// TwinCAT 3 PLC project Untitled1
// ProgramVersion: 3.1.4024.0
// libraries:
//   Tc2_Standard, * (Beckhoff Automation GmbH)
//   Tc2_System, * (Beckhoff Automation GmbH)
//   Tc2_Utilities, * (Beckhoff Automation GmbH)
//   Tc3_Module, * (Beckhoff Automation GmbH)
//   VisuDialogs, * (System)
// project tree:
//   DUTs/ E_PIZZA_TYPES.TcDUT, ST_PIZZA.TcDUT
//   / GlobalTextList.TcGTLO, PlcTask.TcTTO, Visualization Manager.TcVMO (not stored)
//   GVLs/ HMI_VARS.TcGVL
//   POUs/ FB_PizzaOven.TcPOU, F_FIFO_WRITE.TcPOU, MAIN.TcPOU
//   VISUs/ Visualization.TcVIS
// real-time tasks:
//   TASK PlcTask: cycle T#10ms, priority 20, ADS port 350

CONFIGURATION Untitled1
    RESOURCE PLC ON TwinCAT3
        TASK PlcTask(INTERVAL := T#10ms, PRIORITY := 20);
        PROGRAM MAIN WITH PlcTask : MAIN;
    END_RESOURCE
END_CONFIGURATION

// ---- DUTs/E_PIZZA_TYPES.TcDUT
{attribute 'qualified_only'}
{attribute 'strict'}
TYPE E_PIZZA_TYPES :
(
	eType_Cheese := 0,
	eType_Pepperoni := 1,
	eType_Olives := 2
);
END_TYPE

// ---- DUTs/ST_PIZZA.TcDUT
TYPE ST_PIZZA :
STRUCT
	bExist : BOOL;
	dtTimeEnteredOven : DT;
	dtTimeExitedOven : DT;
	tTimeInOven : TIME;
	eType : E_PIZZA_TYPES;	// 0 - cheese, 1 - pepperoni, 2 - olives
END_STRUCT
END_TYPE

// ---- GVLs/HMI_VARS.TcGVL
{attribute 'qualified_only'}
VAR_GLOBAL
	iState : DINT;
	bStartButton : BOOL;
	
	arrPizzaHistory : ARRAY[0..100] OF ST_PIZZA;	
	
	fbNT_GetTime: NT_GetTime;
	stCurrentTime : TIMESTRUCT;
	
END_VAR

// ---- POUs/MAIN.TcPOU
PROGRAM MAIN
VAR
	
	fbMyPizzaOven : ARRAY[0..MAX_OVENS] OF FB_PizzaOven;	// My instance of oven 1
	
	bLoadPizza : BOOL;	// Put a pizza on the input side
	bRemovePizza : BOOL;	// Take pizza off output side
	
	i : DINT;
	
	fbMyTimer : TON;
	
	fbNT_GetTime: NT_GetTime;

END_VAR

VAR CONSTANT
	MAX_OVENS : DINT := 1; // This is 2 because the array starts at 0
END_VAR

FOR i:= 0 TO MAX_OVENS DO
	fbMyPizzaOven[i](bLoadPizza:=bLoadPizza, bRemovePizza:=bRemovePizza);
END_FOR

fbMyTimer(IN:=NOT fbMyTimer.Q, PT:=T#100MS);

fbNT_GetTime(
	NETID := '',
	START := fbMyTimer.Q,
	TIMESTR => hmi_vars.stCurrentTime);

END_PROGRAM

// ---- POUs/FB_PizzaOven.TcPOU
FUNCTION_BLOCK FB_PizzaOven
VAR_INPUT
	
	bLoadPizza : BOOL;	// Put a pizza on the input side
	bRemovePizza : BOOL;	// Take pizza off output side

END_VAR
VAR_OUTPUT

	bBuzzer : BOOL;
	bLight : BOOL;

	iTotalPizzasCooked : UDINT;

END_VAR
VAR
	
	stCurrentTime : TIMESTRUCT;
	dtCurrentTime : DT;

	fbLoad_RTRIG : R_TRIG;
	fbRemove_RTRIG : R_TRIG;	

	stPizzaOnDeck : ST_PIZZA;	// Location of possible pizza
	stPizzaInOven : ST_PIZZA;
	stPizzaDone : ST_PIZZA;
	
	// timers
	fbMyTimer : TON;	// My timer... for stuff.

	iState : DINT;
	ILastState : DINT;
	sStateDesc : STRING;
	arrStateDescHistory : ARRAY[1..100] OF STRING;
	
	bStartButton: BOOL;
	arrPizzaHistory: BYTE;
	TIMESTR: STRING(INT#4);
END_VAR
VAR CONSTANT
	stNULL_PIZZA : ST_PIZZA;
END_VAR

dtCurrentTime := SYSTEMTIME_TO_DT(stCurrentTime);

// If there is room
IF stPizzaOnDeck.bExist AND NOT stPizzaInOven.bExist THEN
	stPizzaInOven := stPizzaOnDeck;
	stPizzaOnDeck := stNULL_PIZZA;	// Remove pizza
END_IF

fbLoad_RTRIG(clk := bLoadPizza);
IF fbLoad_RTRIG.Q THEN
	stPizzaOnDeck.bExist := TRUE;
	stPizzaOnDeck.eType := 2;	// Olives
END_IF

fbRemove_RTRIG(clk := bRemovePizza);
IF fbRemove_RTRIG.Q THEN
	//F_FIFO_WRITE(cbData := SIZEOF(stPizzaDone), pData := ADR(stPizzaDone),
	//				cbBuffer := SIZEOF(arrPizzaHistory), pBuffer := ADR(arrPizzaHistory)
	//);	//It gives an error for arrPizzaHistory, I don't know how to fix it
	stPizzaDone := stNULL_PIZZA;
END_IF

CASE iState OF
	0:	// Wait for pizza in oven
		sStateDesc := 'Waiting on pizza now.';
		IF stPizzaInOven.bExist THEN
			stPizzaInOven.dtTimeEnteredOven := dtCurrentTime;
			iState := 10;
		END_IF
	10:	// We just got a pizza!
		sStateDesc := 'Baking that pizza now.';
		fbMyTimer(IN:=TRUE, PT:=T#3S);
		
		IF fbMyTimer.Q THEN
			fbMyTimer(IN:=FALSE);
			iState := 20;
		END_IF
	20:	// Can we move the pizza out of the oven? It's going to burn!
		IF NOT stPizzaDone.bExist THEN
			// Simulate conveyor
			stPizzaInOven.dtTimeExitedOven := dtCurrentTime;
			stPizzaDone := stPizzaInOven;
			stPizzaInOven := stNULL_PIZZA;
			bBuzzer := FALSE;
			iState := 30;
		ELSE
			bBuzzer := TRUE;
			sStateDesc := 'The pizza is burning!';
		END_IF
	30:	// Pizza just removed on output tray
		stPizzaInOven.tTimeInOven := stPizzaInOven.dtTimeExitedOven - stPizzaInOven.dtTimeEnteredOven;
		iTotalPizzasCooked := iTotalPizzasCooked + 1;
		iState := 0;	// Go wait for new pizza in oven!
ELSE
	sStateDesc := 'Invalid state!';
END_CASE

// Start state history

IF iLastState <> iState THEN
	// Do stuff here to log transitions...
	F_FIFO_WRITE(cbData := SIZEOF(sStateDesc), pData := ADR(sStateDesc),
					cbBuffer := SIZEOF(arrStateDescHistory), pBuffer := ADR(arrStateDescHistory)
	);
	// ^^ SIZEOF returns the count in bytes
	
	// Reset for next time
	iLastState := iState;
END_IF

END_FUNCTION_BLOCK

// ---- POUs/F_FIFO_WRITE.TcPOU
FUNCTION F_FIFO_WRITE : BOOL
VAR_INPUT
	cbData : UDINT;	// Stuff coming in (length of one data element)
	pData : POINTER TO BYTE;
	
	cbBuffer : UDINT;	// Where all the stuff lives
	pBuffer : POINTER TO BYTE;	// first bit
END_VAR
VAR
END_VAR

// Logic behind pDest, pBuffer tells us where we are in the memory, cbData tells us the type,
// for example if it's a UDINT then cbData is gonna be 4 bytes, so if we add up where we are and cbData,
// we get where we wanna be
FW_MemMove(pDest := pBuffer + cbData, pSrc := pBuffer, cbLen := cbBuffer - cbData);	
// ^^ Take everything and move it down (memory wise)

FW_MemMove(pDest := pBuffer, pSrc := pData, cbLen := cbData);
// ^^ Place in the first row (memory wise) - user provided

END_FUNCTION

// ---- GlobalTextList.TcGTLO
TEXTLIST GlobalTextList
  804 = 'B'
  935 = 'Buzzer'
  182 = 'Elapsed Time:'
  112 = 'Elapsed Time: %s'
  972 = 'Insert Pizza'
  202 = 'L'
  596 = 'Light'
  614 = 'New Pizza Ready'
  452 = 'Package Pizza'
  356 = 'Pizza'
  333 = 'Pizza (Done)'
  889 = 'Pizza (On Deck)'
  679 = 'Pizzas Cooked: %d'
  153 = 'Status: %d'
  405 = 'Status: %s'
  635 = 'Take Pizza Out'
END_TEXTLIST

// ---- VISUs/Visualization.TcVIS
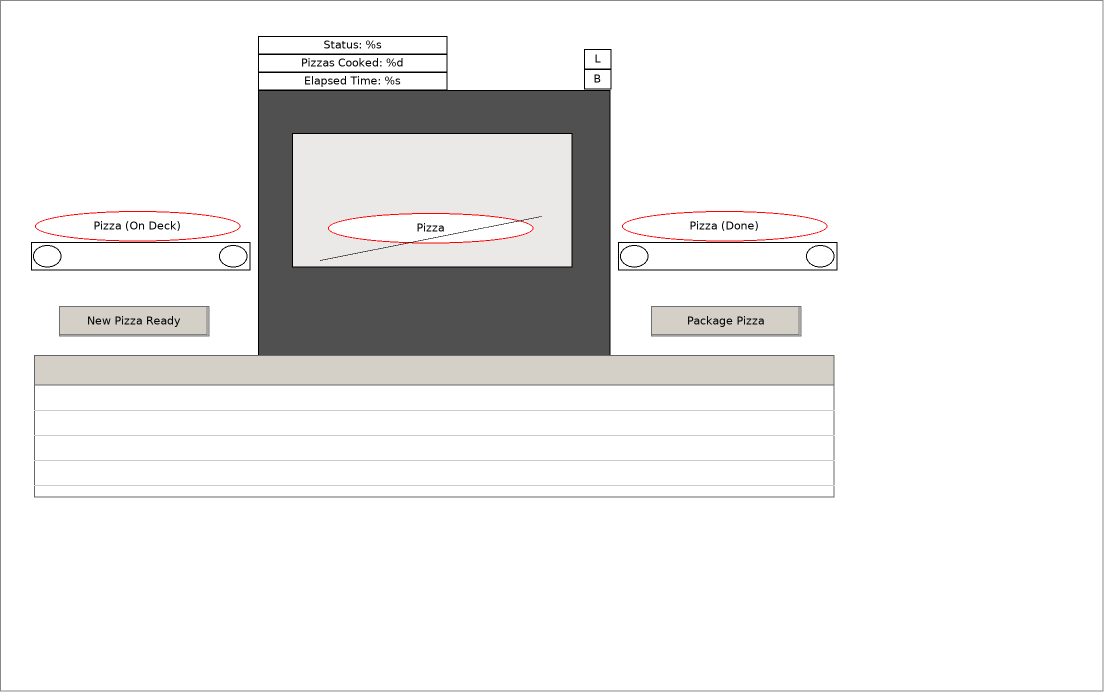
VISUALIZATION Visualization  // 1104x692
    Line (1103,691)
    Rectangle (258,90 352x366)
    Button (59,306 150x30), "New Pizza Ready"
        tap MAIN.bLoadPizza
    Button (651,306 150x30), "Package Pizza"
        tap MAIN.bRemovePizza
    Rectangle (292,133 280x134)
    Ellipse (328,213 205x30), "Pizza", invisible if: NOT MAIN.fbMyPizzaOven[0].stPizzaInOven.bExist
    Rectangle (258,72 189x18), "Elapsed Time: %s", text variable: Main.fbMyPizzaOven[0].fbMyTimer.ET
    Line (320,260) (541,216)
    Rectangle (258,54 189x18), "Pizzas Cooked: %d", text variable: MAIN.fbMyPizzaOven[0].iTotalPizzasCooked
    RoundedRectangle (584,69 27x20), "B", colour toggle: Main.fbMyPizzaOven[0].bBuzzer
    RoundedRectangle (584,49 27x20), "L"
    Rectangle (31,242 219x28)
    Ellipse (35,211 205x30), "Pizza (On Deck)", invisible if: NOT Main.fbMyPizzaOven[0].stPizzaOnDeck.bExist
    Ellipse (33,245 28x22)
    Ellipse (219,245 28x22)
    Rectangle (618,242 219x28)
    Ellipse (622,211 205x30), "Pizza (Done)", invisible if: NOT Main.fbMyPizzaOven[0].stPizzaDone.bExist
    Ellipse (620,245 28x22)
    Ellipse (806,245 28x22)
    Rectangle (258,36 189x18), "Status: %s", text variable: MAIN.fbMyPizzaOven[0].sStateDesc
    Table (34,355 800x142), data array: HMI_VARS.arrPizzaHistory
        p3854506369: HMI_VARS.arrPizzaHistory[INDEX].bExist
        p1892666644: HMI_VARS.arrPizzaHistory[INDEX].dtTimeEnteredOven
        p338671338: HMI_VARS.arrPizzaHistory[INDEX].dtTimeExitedOven
        p2170511999: HMI_VARS.arrPizzaHistory[INDEX].tTimeInOven
        p3723444502: HMI_VARS.arrPizzaHistory[INDEX].eType
END_VISUALIZATION
